TYPE "SpeedMotor_Config"
VERSION : 0.1
// Block: SpeedMotor_Config
   STRUCT
      ReferenceVelocity : LReal;
      InvertDirection : Bool;
   END_STRUCT;

END_TYPE
